{attribute addProperty BoxType "EL1512-0000-0016"}
{attribute addProperty Id "Set_counter_doneAT %I*BOOL813Counter_inhibitedAT %I*BOOL814Status_of_input_clockAT %I*BOOL816TxPDO_ToggleAT %I*BOOL819Counter_valueAT %I*UDINT32417"}
{attribute addProperty CRC "1146763198"}
{attribute addProperty SizeInBites "64"}
{attribute addProperty SizeInBytes "8"}
TYPE CNT_Inputs_Channel_445A37BE :
STRUCT
	{attribute addProperty Name "Set_counter_done"}
	Set_counter_done AT %I* : BOOL;
	{attribute addProperty Name "Counter_inhibited"}
	Counter_inhibited AT %I* : BOOL;
	{attribute addProperty Name "Status_of_input_clock"}
	Status_of_input_clock AT %I* : BOOL;
	{attribute addProperty Name "TxPDO_Toggle"}
	TxPDO_Toggle AT %I* : BOOL;
	{attribute addProperty Name "Counter_value"}
	Counter_value AT %I* : UDINT;
END_STRUCT
END_TYPE

(* stored: Version 1.2.0.0, ProductVersion 3.1.4024.9
   DUT CNT_Inputs_Channel_445A37BE: Id {80afbb35-5d75-4054-b087-187576f14a84} *)
